FUNCTION_BLOCK FB_AxisStatusNC_TestDouble IMPLEMENTS I_AxisStatus
VAR
	bError : BOOL;
	nErrorID : UDINT := 24000;
END_VAR

{warning 'Add property implementation'}
PROPERTY Aborted : BOOL
GET
END_GET
END_PROPERTY

{warning 'Add property implementation'}
PROPERTY Active : BOOL
GET
END_GET
END_PROPERTY

{warning 'Add method implementation '}
METHOD AxisEnabled : BOOL
END_METHOD

{warning 'Add property implementation'}
PROPERTY AxisID : UDINT
GET
END_GET
END_PROPERTY

{warning 'Add property implementation'}
PROPERTY AxisState : MC_AxisStates
GET
END_GET
END_PROPERTY

{warning 'Add property implementation'}
PROPERTY Busy : BOOL
GET
END_GET
END_PROPERTY

{warning 'Add property implementation'}
PROPERTY Done : BOOL
GET
END_GET
END_PROPERTY

{warning 'Add property implementation'}
PROPERTY Error : BOOL
GET
Error := bError;
END_GET
SET
bError := Error;
END_SET
END_PROPERTY

{warning 'Add property implementation'}
PROPERTY ErrorID : UDINT
GET
ErrorId := nErrorID;
END_GET
SET
nErrorId := ErrorID;
END_SET
END_PROPERTY

{warning 'Add property implementation'}
PROPERTY InTargetPosition : BOOL
GET
END_GET
END_PROPERTY

{warning 'Add property implementation'}
PROPERTY MeasuredAcceleration : LREAL
GET
END_GET
END_PROPERTY

{warning 'Add property implementation'}
PROPERTY MeasuredPosition : LREAL
GET
END_GET
END_PROPERTY

{warning 'Add property implementation'}
PROPERTY MeasuredPositionDiff : LREAL
GET
END_GET
END_PROPERTY

{warning 'Add property implementation'}
PROPERTY MeasuredVelocity : LREAL
GET
END_GET
END_PROPERTY

{warning 'Add property implementation'}
PROPERTY Message : T_MAXSTRING
GET
END_GET
END_PROPERTY

{warning 'Add property implementation'}
PROPERTY NegativeMotionIsEnabled : BOOL
GET
END_GET
END_PROPERTY

{warning 'Add property implementation'}
PROPERTY PositiveMotionIsEnabled : BOOL
GET
END_GET
END_PROPERTY

{warning 'Add property implementation'}
PROPERTY StandStill : BOOL
GET
END_GET
END_PROPERTY

{warning 'Add property implementation'}
PROPERTY Stopped : BOOL
GET
END_GET
END_PROPERTY

END_FUNCTION_BLOCK

(* stored: Version 1.1.0.1
   POU FB_AxisStatusNC_TestDouble: Id {3bc600b5-957e-4849-b712-96877efc6ba9}, SpecialFunc None
   Property Aborted: Id {cc170558-0620-458d-87a8-699df73a8a75}
   Get Get: Id {f9f1e2c4-d8a9-45ce-9909-19b7af0a1cbb}
   Property Active: Id {7a35bbf9-afb3-4d08-bdce-aeb177c8e552}
   Get Get: Id {08e90f8d-49b8-4c06-bc19-b845a403e3e0}
   Method AxisEnabled: Id {4fe0c85f-bfea-44c4-a30e-3d6a1e0c191a}
   Property AxisID: Id {4dd060ea-90f2-42d9-bcbf-23403d3dc094}
   Get Get: Id {4c027711-f1f9-4068-a2f8-3b95309c82f6}
   Property AxisState: Id {0d9ad659-80bd-4f63-b9ca-93106f3ede20}
   Get Get: Id {2db314fc-2e98-4971-9c34-3337a8d32d7f}
   Property Busy: Id {9d678886-9e63-4f4e-87cc-525b5e515ae6}
   Get Get: Id {c936cd76-a12e-43f7-8687-07613827f9ca}
   Property Done: Id {92666856-d948-4698-a58b-0fd925a9db1b}
   Get Get: Id {c7f70d5f-1ef9-48b4-9571-62c385faf274}
   Property Error: Id {67a362a3-5d8c-4e59-9895-d93673d24cf3}
   Get Get: Id {443656d5-3f6a-45bb-b2ba-6be9780557c1}
   Set Set: Id {b54ff63e-3a41-41f8-852f-1028d4fea4b8}
   Property ErrorID: Id {5293159e-8ec9-497b-b441-e3920999203e}
   Get Get: Id {c432912c-6068-440d-a8ef-7a54f2b6ca5e}
   Set Set: Id {6db9fc17-d098-4b71-9fbd-ed3f9ba1a8de}
   Property InTargetPosition: Id {5e227f4c-263b-4939-bdd2-6bd10935d1be}
   Get Get: Id {f12c499c-c553-41cc-86b2-f482cfcd10fc}
   Property MeasuredAcceleration: Id {e69d6f11-8d2c-4b72-b569-ad94a043dbcb}
   Get Get: Id {98476150-8466-4f78-a084-26619cab0301}
   Property MeasuredPosition: Id {cc2bbd09-aa9a-497c-93f1-285f68d6247a}
   Get Get: Id {2a8953b9-edc7-4df0-9e52-bc867615f820}
   Property MeasuredPositionDiff: Id {dc8f2aa8-1e3e-4b68-93f0-dc4ae6c3156d}
   Get Get: Id {693d24e4-92c8-46a1-9321-6db2dcc4ae6a}
   Property MeasuredVelocity: Id {92a90de6-385e-409d-a64d-c620fd40a957}
   Get Get: Id {72a27b52-8a28-4fd8-838b-0897360bd680}
   Property Message: Id {88a29df3-3a2c-45ef-ba32-e169ad9b053e}
   Get Get: Id {b1cf1ef3-3cf4-4cc3-8cac-60d6e2ca30b5}
   Property NegativeMotionIsEnabled: Id {60f1a34e-31a0-4d7c-b94c-f2d787a96c65}
   Get Get: Id {4281da51-879d-4b65-84ae-956219c721c4}
   Property PositiveMotionIsEnabled: Id {f9ae3098-56b9-4003-a867-b5a73ad4fe63}
   Get Get: Id {c5436c6e-2a5b-4640-aa30-377de879990c}
   Property StandStill: Id {ab318470-bff5-48c7-b910-d942672f236a}
   Get Get: Id {51937155-75ec-4830-85ec-5e796a600f5d}
   Property Stopped: Id {546d7abb-0fb3-4853-bded-69b1f1724c12}
   Get Get: Id {bc18d421-91a5-44f6-b15c-87fee8794138} *)
